PROGRAM PRG_SavePeristentVariables
VAR
    fbWritePersistentData: FB_WritePersistentData;
    tonStart : TON;
    tonInterval : TON;
END_VAR

tonInterval(
    IN:=TRUE,
    PT:=T#1ms (* Write 1ms after startup of the PLC *)

);

tonStart(
    IN:=tonStart.Q AND NOT fbWritePersistentData.BUSY,
    PT:=T#1m (* Write every minute *)
);

fbWritePersistentData(
    NETID:='', (* This PLC *)
    PORT:=851, (* Application port! *)
    TMOUT:=T#10s,  (* Maximum time before considering this a failure *)
    START:=tonStart.Q OR tonInterval.Q (* Start with tonStart goes high or periodically *)
);

END_PROGRAM

(* stored: Version 1.1.0.1, ProductVersion 3.1.4022.18
   POU PRG_SavePeristentVariables: Id {df16ef79-2907-4ff9-80ce-e27d47a4e69d}, SpecialFunc None *)
